// TIA Portal V21 export
DATA_BLOCK "Zona"   // DB26
{ S7_Optimized_Access := 'TRUE' }
// stored: MemoryReserve 100
   VAR RETAIN
      Comuni : Struct
         ResetFromHMI : Bool := FALSE;
         TempoCicloCpu_r : Real := 0.1030251;
         Clocks : Struct
            Clock1Hz : Bool := TRUE;
            Clock1Hz_Memo : Bool := TRUE;   // Stato precedente
            "Clock0.2Hz" : Bool := TRUE;
            "Clock0.2Hz_Memo" : Bool := TRUE;
            RuntimeClock : LReal := 16#0002_CA53_7981_7592;
            TempoPassato : LReal := 0.0;
         END_STRUCT;
         AlmenoUnaZonaInUpdate : Bool := TRUE;   // Almeno una zona in update
         UpdateGenerale : Bool := FALSE;   // Update di tutto il software
         Login : Struct
            UtenteAttuale : Struct
               Livello : Int := 0;
               Numero : Int := 0;
               Timeout : "Std_stTimer";
            END_STRUCT;
            Lista : Array[0.."K_NumUtente"] of "Std_Utente";
            Hmi : Struct
               Richiesto : "Std_Utente";
               Comandi : Struct
                  Login : Bool := FALSE;
                  Logout : Bool := FALSE;
               END_STRUCT;
            END_STRUCT;
         END_STRUCT;
         TempoCicloProgramma : Struct
            AppoTempoCiclo : LReal := 0.0;
            DatiUtili : "Std_TCiclo";
            Login : "Std_TCiclo";
            Motori : "Std_TCiclo";
            Valvole : "Std_TCiclo";
            Analogiche : "Std_TCiclo";
            Zone : "Std_TCiclo";
            Sequenze : "Std_TCiclo";
            Ricette : "Std_TCiclo";
            Popups : "Std_TCiclo";
            Tot : Struct
               Act : LReal := 0.0;
               PercTciclo : Real := 0.0;
               Prec : LReal := 0.0;
            END_STRUCT;
         END_STRUCT;
         Simulazione_PLCSim : Bool := FALSE;
         "1HzCount++" : Int := 17;   // Numero che incrementa ogni mezzo secondo
         "0.20HzCount++" : Int := 4;   // Numero che incrementa ogni decimo di secondo
         FirstScanFromCpu : Bool := FALSE;
      END_STRUCT;
   END_VAR
   VAR
      DiagnosticaProgrammatore : Struct
         Comandi : Struct
            AbilitaDiagnosticaProgrammatore : Bool := FALSE;
            ResettaAllarmi : Bool := FALSE;
         END_STRUCT;
         ErroriRichiami : Array[0.."K_NumKTipo"] of Struct
            LimiteArraySuperato : Struct
               Stato : Bool;   // Indica se il limitre dell'array è stato superato
               "Da(Tipo)" : Int;   // Indica quale tipo di utenza sbaglia a puntare all'array
               "Num(Indice)" : Int;   // Indica il numero dell'utenza che sbaglia
            END_STRUCT;
            MultiRichiamo : Struct
               Allarme : Bool;
               TipoUtenza : Int;   // Indica quale tipo di utenza sbaglia a puntare all'array
               IndiceUtenza : Int;   // Indica il numero dell'utenza che sbaglia
            END_STRUCT;
         END_STRUCT;
         LimiteArraySuperato : Struct   // Verificare l'accesso nell'array
            Stato : Bool := FALSE;   // Indica se il limitre dell'array è stato superato
            "Da(Tipo)" : Int := 0;   // Indica quale tipo di utenza sbaglia a puntare all'array
            "Num(Indice)" : Int := 0;   // Indica il numero dell'utenza che sbaglia
         END_STRUCT;
      END_STRUCT;
   END_VAR
   VAR RETAIN
      Z : Array[0.."K_NumZona"] of "Std_Zona";
   END_VAR
BEGIN
   Comuni.Login.UtenteAttuale.Timeout.IN := FALSE;
   Comuni.Login.UtenteAttuale.Timeout.O := FALSE;
   Comuni.Login.UtenteAttuale.Timeout.Preset := 0.0;
   Comuni.Login.UtenteAttuale.Timeout.TempoTrascorso := 0.0;
   Comuni.Login.Lista[0].User := '';
   Comuni.Login.Lista[0].Psw := '';
   Comuni.Login.Lista[0].Livello := 0;
   Comuni.Login.Lista[0].TimeOut := 0.0;
   Comuni.Login.Hmi.Richiesto.User := '';
   Comuni.Login.Hmi.Richiesto.Psw := '';
   Comuni.Login.Hmi.Richiesto.Livello := 0;
   Comuni.Login.Hmi.Richiesto.TimeOut := 0.0;
   Comuni.TempoCicloProgramma.DatiUtili.Act := 0.0;
   Comuni.TempoCicloProgramma.DatiUtili.PercTciclo := 0.0;
   Comuni.TempoCicloProgramma.Login.Act := 0.0;
   Comuni.TempoCicloProgramma.Login.PercTciclo := 0.0;
   Comuni.TempoCicloProgramma.Motori.Act := 0.0;
   Comuni.TempoCicloProgramma.Motori.PercTciclo := 0.0;
   Comuni.TempoCicloProgramma.Valvole.Act := 0.0;
   Comuni.TempoCicloProgramma.Valvole.PercTciclo := 0.0;
   Comuni.TempoCicloProgramma.Analogiche.Act := 0.0;
   Comuni.TempoCicloProgramma.Analogiche.PercTciclo := 0.0;
   Comuni.TempoCicloProgramma.Zone.Act := 0.0;
   Comuni.TempoCicloProgramma.Zone.PercTciclo := 0.0;
   Comuni.TempoCicloProgramma.Sequenze.Act := 0.0;
   Comuni.TempoCicloProgramma.Sequenze.PercTciclo := 0.0;
   Comuni.TempoCicloProgramma.Ricette.Act := 0.0;
   Comuni.TempoCicloProgramma.Ricette.PercTciclo := 0.0;
   Comuni.TempoCicloProgramma.Popups.Act := 0.0;
   Comuni.TempoCicloProgramma.Popups.PercTciclo := 0.0;
   DiagnosticaProgrammatore.ErroriRichiami[0..16].LimiteArraySuperato.Stato := FALSE;
   DiagnosticaProgrammatore.ErroriRichiami[0..16].LimiteArraySuperato."Da(Tipo)" := 0;
   DiagnosticaProgrammatore.ErroriRichiami[0..16].LimiteArraySuperato."Num(Indice)" := 0;
   DiagnosticaProgrammatore.ErroriRichiami[0..16].MultiRichiamo.Allarme := FALSE;
   DiagnosticaProgrammatore.ErroriRichiami[0..16].MultiRichiamo.TipoUtenza := 0;
   DiagnosticaProgrammatore.ErroriRichiami[0..16].MultiRichiamo.IndiceUtenza := 0;
   // DiagnosticaProgrammatore.ErroriRichiami[1] : K_TipoAnalogica
   // DiagnosticaProgrammatore.ErroriRichiami[2] : K_TipoPid
   // DiagnosticaProgrammatore.ErroriRichiami[3] : K_TipoMisuratoreFlusso
   // DiagnosticaProgrammatore.ErroriRichiami[4] : K_TipoTrend
   // DiagnosticaProgrammatore.ErroriRichiami[5] : K_TipoParatia
   // DiagnosticaProgrammatore.ErroriRichiami[6] : K_TipoMotore
   // DiagnosticaProgrammatore.ErroriRichiami[7] : K_TipoPompa
   // DiagnosticaProgrammatore.ErroriRichiami[8] : K_TipoValvola
   // DiagnosticaProgrammatore.ErroriRichiami[9] : K_TipoSezionePastorizzatore
   // DiagnosticaProgrammatore.ErroriRichiami[10] : K_TipoZona
   // DiagnosticaProgrammatore.ErroriRichiami[11] : K_TipoComunicazione
   // DiagnosticaProgrammatore.ErroriRichiami[12] : K_TipoSequenza
   // DiagnosticaProgrammatore.ErroriRichiami[13] : K_TipoSegnaliMacchine
   // DiagnosticaProgrammatore.ErroriRichiami[14] : K_TipoSensore
   Z[0].In.RichiestaLampadaReset := TRUE;
   Z[0].Gen.UpdatePrm_Mem := FALSE;
   Z[0].Gen.UpdatePrm := TRUE;
   Z[0].Gen.ResetLoc_Hmi := FALSE;
   Z[0].Gen.Reset := FALSE;
   Z[0].Prm.CentralinaOkDaTempo.IN := FALSE;
   Z[0].Prm.CentralinaOkDaTempo.O := FALSE;
   Z[0].Prm.CentralinaOkDaTempo.Preset := 1.0;
   Z[0].Prm.CentralinaOkDaTempo.TempoTrascorso := 0.0;
   Z[0].Prm.RitardoCicloAuto.IN := FALSE;
   Z[0].Prm.RitardoCicloAuto.O := FALSE;
   Z[0].Prm.RitardoCicloAuto.Preset := 1.0;
   Z[0].Prm.RitardoCicloAuto.TempoTrascorso := 0.0;
   Z[0].Prm.RitardoCicloMan.IN := FALSE;
   Z[0].Prm.RitardoCicloMan.O := FALSE;
   Z[0].Prm.RitardoCicloMan.Preset := 1.0;
   Z[0].Prm.RitardoCicloMan.TempoTrascorso := 0.0;
   Z[0].Prm.RitardoStopDaTempo.IN := FALSE;
   Z[0].Prm.RitardoStopDaTempo.O := FALSE;
   Z[0].Prm.RitardoStopDaTempo.Preset := 0.0;
   Z[0].Prm.RitardoStopDaTempo.TempoTrascorso := 0.0;
   Z[0].Dati.BloccoRichiamato := FALSE;
   Z[0].Allarmi.Prm.PulisciStoricoUtenze := FALSE;
   Z[0].Allarmi.SlotAllarmeDaUtenze[0..5].Allarme := FALSE;
   Z[0].Allarmi.SlotAllarmeDaUtenze[0..5].AllarmeSilenziato := FALSE;
   Z[0].Allarmi.SlotAllarmeDaUtenze[0..5].TipoNum := 0;
   Z[0].Allarmi.SlotAllarmeDaUtenze[0].TipoNome := '';
   Z[0].Allarmi.SlotAllarmeDaUtenze[1].TipoNome := 'Motore';
   Z[0].Allarmi.SlotAllarmeDaUtenze[2..5].TipoNome := '';
   Z[0].Allarmi.SlotAllarmeDaUtenze[0..5].Indice := 0;
   Z[0].Allarmi.SlotAllarmeDaUtenze[0..5].NumAllarme := 0;
   Z[0].Allarmi."A"[0..13].Abilitato := FALSE;
   Z[0].Allarmi."A"[0..13].Stato := FALSE;
   Z[0].Allarmi."A"[0..13].Silenziato := FALSE;
   Z[0].Allarmi."A"[0].EnWarnHmi := FALSE;
   Z[0].Allarmi."A"[1..2].EnWarnHmi := TRUE;
   Z[0].Allarmi."A"[3..13].EnWarnHmi := FALSE;
   Z[0].Allarmi."A"[0].EnCadutaCiclo := FALSE;
   Z[0].Allarmi."A"[1..2].EnCadutaCiclo := TRUE;
   Z[0].Allarmi."A"[3..13].EnCadutaCiclo := FALSE;
   Z[0].Allarmi.AG[0..15].Abilitato := FALSE;
   Z[0].Allarmi.AG[0..15].Stato := FALSE;
   Z[0].Allarmi.AG[0..15].Silenziato := FALSE;
   Z[0].Allarmi.AG[0..15].EnWarnHmi := FALSE;
   Z[0].Allarmi.AG[0..15].EnCadutaCiclo := FALSE;
   Z[0].Allarmi.WordHMI := 16#0000;
   Z[0].Allarmi.WordHMI_AG := 16#0000;
   Z[0].Out.Auto := FALSE;
   Z[0].Out.Man := FALSE;
   Z[0].Out.Attivo := FALSE;
   Z[0].Out.StopDaTempo := TRUE;
   Z[0].Out.Attesa := FALSE;
   Z[0].Out.AutoDaHmi := FALSE;
   Z[0].Out.Stato := 0;
   Z[0].Out.CumulativoAllarmi := FALSE;
   Z[0].Out.SirenaSuona := TRUE;
   Z[0].Out.CentralinaOk := FALSE;
   Z[0].Rif_Inc.K_Zona_Padre := 0;
END_DATA_BLOCK
